(* CoDeSys 2.3.9.42 project: Preobrazovatel_84.pro *)

(* POU PLC_PRG, ST *)
PROGRAM PLC_PRG
VAR
	tok_low:REAL:=4;
	tok_high:REAL:=20;
	diap_low,diap_high :REAL; (*диапазоны измеряемой температуры *)
	Tok : REAL ; (*ток 4-20 мА*)
	Prom : REAL ; (*промежеточная переменная*)
	lamp_yellow: BOOL; (*лампа, выход за диапазон градусов*)
	Temperatura: REAL; (*температура*)
END_VAR
lamp_yellow := (Tok > tok_high) OR (Tok < tok_low) ;

Prom:=LIMIT(tok_low, Tok, tok_high);

Temperatura:=((diap_high*(Prom-4))/16);


preobra;
END_PROGRAM

(* POU preobra, CFC *)
PROGRAM preobra
VAR
	Tok: REAL;
	tok_high: REAL;
	tok_low: REAL;
	lamp_yellow: BOOL;
END_VAR
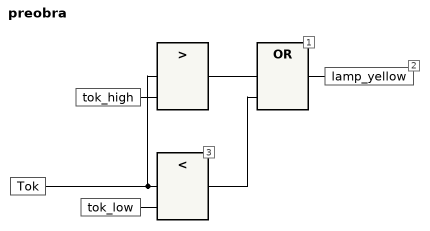
_CFC_ (* Continuous Function Chart, elements in execution order *)
#0 >(Tok, tok_high)
#1 OR(#0, #3)
#2 lamp_yellow <= #1
#3 <(Tok, tok_low)
_END_CFC_
END_PROGRAM
